FUNCTION_BLOCK FB_TurnControlEmulation 
VAR_INPUT	
	Config					: ST_CFG_TurnTablePositionEmu; // emulation config	
	DriveRun_CW			: BOOL;
	DriveRun_CCW        : BOOL;
END_VAR

VAR_OUTPUT
	Turn_Pos_CW				: BOOL;
	Turn_Pos_CCW			: BOOL;
	Turn_Pos_Middle_CW		: BOOL;
	Turn_Pos_Middle_CCW		: BOOL;
END_VAR

VAR
	ActualPosition			: INT :=0;
END_VAR



// When lift is moving
IF DriveRun_CW THEN
	IF ActualPosition < Config.Position_Max_CW THEN
	ActualPosition := ActualPosition + 1;
	END_IF
END_IF

IF DriveRun_CCW THEN
	IF ActualPosition > Config.Position_Max_CCW THEN
	ActualPosition := ActualPosition - 1;
	END_IF
END_IF


// Update positions
IF ActualPosition = Config.Position_CCW THEN
	 Turn_Pos_CCW := TRUE;
ELSIF ActualPosition = Config.Position_CW THEN
	 Turn_Pos_CW := TRUE;
ELSIF ActualPosition = Config.Position_Middle_CW THEN
	Turn_Pos_Middle_CW := TRUE;
	Turn_Pos_Middle_CCW := TRUE;

(* Debug code for emulating creep. since the Positions may be changed in project configuration, this is disabled to reduce risk of emulation error
ELSIF ActualPosition < Config.Position_Middle_CW AND ActualPosition > Config.Position_Middle_CW-30 THEN //Turning from CCW
	Turn_Pos_Middle_CW := FALSE;
	Turn_Pos_Middle_CCW := TRUE;
ELSIF ActualPosition > Config.Position_Middle_CW AND ActualPosition < Config.Position_Middle_CW+30 THEN // turning from CW
	Turn_Pos_Middle_CW := FALSE;
	Turn_Pos_Middle_CCW := TRUE;
*)
ELSE  	
	Turn_Pos_CCW := FALSE;
	Turn_Pos_CW := FALSE;
	Turn_Pos_Middle_CW := FALSE;
	Turn_Pos_Middle_CCW := FALSE;		
END_IF

END_FUNCTION_BLOCK

(* stored: Version 1.1.0.1, ProductVersion 3.1.4024.9
   POU FB_TurnControlEmulation: Id {898a668c-0f8a-42dd-ad86-3b4b1f727e74}, SpecialFunc None *)
